# EPICS substitutions: support/ebrick/2-2-3/iocBoot/iocebrick/ebrickRMMDIF.substitutions
file ../../db/ebrDAC.db
{
pattern
{P         H       F       D       PREC    CH  MIN     MAX     PORT}

{ebrick:   rmm01:  ana01:  ao01    3       0   -10     10      RMMDIF}
{ebrick:   rmm01:  ana01:  ao02    3       2   -10     10      RMMDIF}

}
